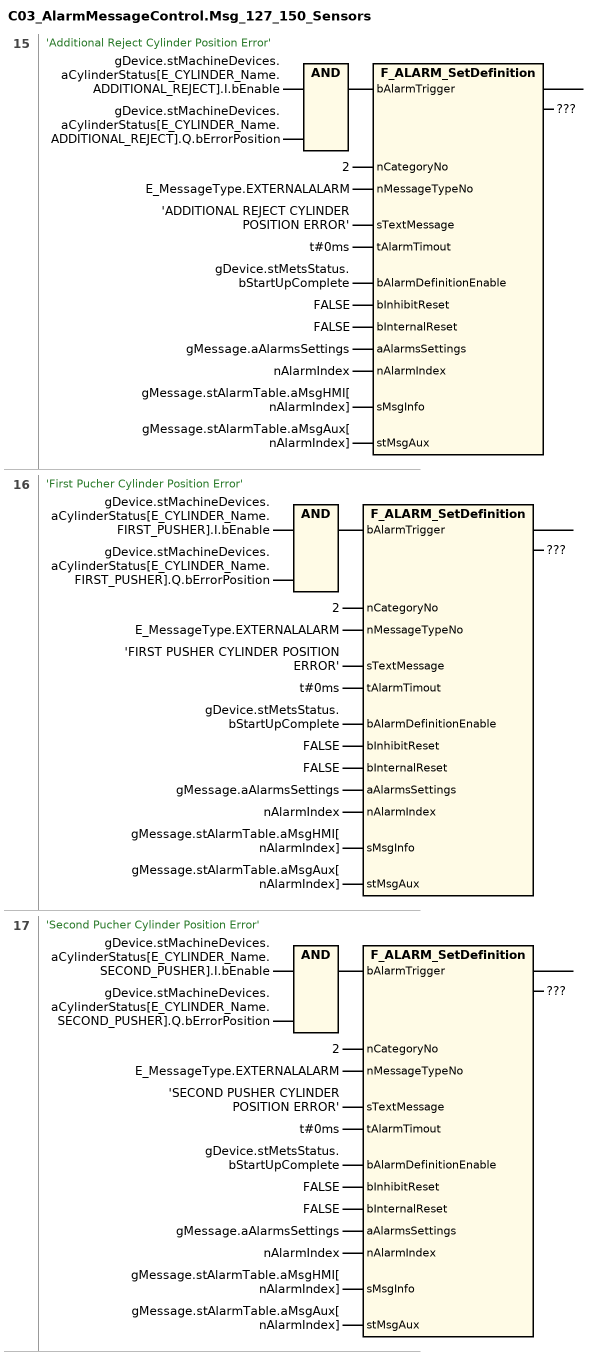
// NETWORK 15
// 'Additional Reject Cylinder Position Error'
F_ALARM_SetDefinition(bAlarmTrigger := gDevice.stMachineDevices.aCylinderStatus[E_CYLINDER_Name.ADDITIONAL_REJECT].I.bEnable AND gDevice.stMachineDevices.aCylinderStatus[E_CYLINDER_Name.ADDITIONAL_REJECT].Q.bErrorPosition, nCategoryNo := 2, nMessageTypeNo := E_MessageType.EXTERNALALARM, sTextMessage := 'ADDITIONAL REJECT CYLINDER POSITION ERROR', tAlarmTimout := t#0ms, bAlarmDefinitionEnable := gDevice.stMetsStatus.bStartUpComplete, bInhibitReset := FALSE, bInternalReset := FALSE, aAlarmsSettings := gMessage.aAlarmsSettings, nAlarmIndex := nAlarmIndex, sMsgInfo := gMessage.stAlarmTable.aMsgHMI[nAlarmIndex], stMsgAux := gMessage.stAlarmTable.aMsgAux[nAlarmIndex]);

// NETWORK 16
// 'First Pucher Cylinder Position Error'
F_ALARM_SetDefinition(bAlarmTrigger := gDevice.stMachineDevices.aCylinderStatus[E_CYLINDER_Name.FIRST_PUSHER].I.bEnable AND gDevice.stMachineDevices.aCylinderStatus[E_CYLINDER_Name.FIRST_PUSHER].Q.bErrorPosition, nCategoryNo := 2, nMessageTypeNo := E_MessageType.EXTERNALALARM, sTextMessage := 'FIRST PUSHER CYLINDER POSITION ERROR', tAlarmTimout := t#0ms, bAlarmDefinitionEnable := gDevice.stMetsStatus.bStartUpComplete, bInhibitReset := FALSE, bInternalReset := FALSE, aAlarmsSettings := gMessage.aAlarmsSettings, nAlarmIndex := nAlarmIndex, sMsgInfo := gMessage.stAlarmTable.aMsgHMI[nAlarmIndex], stMsgAux := gMessage.stAlarmTable.aMsgAux[nAlarmIndex]);

// NETWORK 17
// 'Second Pucher Cylinder Position Error'
F_ALARM_SetDefinition(bAlarmTrigger := gDevice.stMachineDevices.aCylinderStatus[E_CYLINDER_Name.SECOND_PUSHER].I.bEnable AND gDevice.stMachineDevices.aCylinderStatus[E_CYLINDER_Name.SECOND_PUSHER].Q.bErrorPosition, nCategoryNo := 2, nMessageTypeNo := E_MessageType.EXTERNALALARM, sTextMessage := 'SECOND PUSHER CYLINDER POSITION ERROR', tAlarmTimout := t#0ms, bAlarmDefinitionEnable := gDevice.stMetsStatus.bStartUpComplete, bInhibitReset := FALSE, bInternalReset := FALSE, aAlarmsSettings := gMessage.aAlarmsSettings, nAlarmIndex := nAlarmIndex, sMsgInfo := gMessage.stAlarmTable.aMsgHMI[nAlarmIndex], stMsgAux := gMessage.stAlarmTable.aMsgAux[nAlarmIndex]);

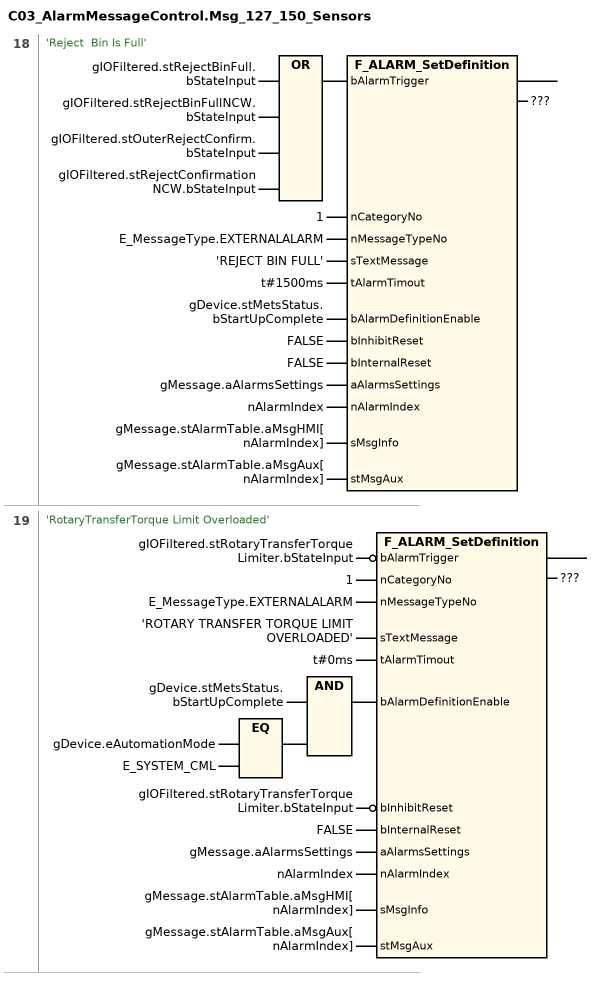
// NETWORK 18
// 'Reject  Bin Is Full'
F_ALARM_SetDefinition(bAlarmTrigger := gIOFiltered.stRejectBinFull.bStateInput OR gIOFiltered.stRejectBinFullNCW.bStateInput OR gIOFiltered.stOuterRejectConfirm.bStateInput OR gIOFiltered.stRejectConfirmationNCW.bStateInput, nCategoryNo := 1, nMessageTypeNo := E_MessageType.EXTERNALALARM, sTextMessage := 'REJECT BIN FULL', tAlarmTimout := t#1500ms, bAlarmDefinitionEnable := gDevice.stMetsStatus.bStartUpComplete, bInhibitReset := FALSE, bInternalReset := FALSE, aAlarmsSettings := gMessage.aAlarmsSettings, nAlarmIndex := nAlarmIndex, sMsgInfo := gMessage.stAlarmTable.aMsgHMI[nAlarmIndex], stMsgAux := gMessage.stAlarmTable.aMsgAux[nAlarmIndex]);

// NETWORK 19
// 'RotaryTransferTorque Limit Overloaded'
F_ALARM_SetDefinition(bAlarmTrigger := NOT gIOFiltered.stRotaryTransferTorqueLimiter.bStateInput, nCategoryNo := 1, nMessageTypeNo := E_MessageType.EXTERNALALARM, sTextMessage := 'ROTARY TRANSFER TORQUE LIMIT OVERLOADED', tAlarmTimout := t#0ms, bAlarmDefinitionEnable := gDevice.stMetsStatus.bStartUpComplete AND gDevice.eAutomationMode = E_SYSTEM_CML, bInhibitReset := NOT gIOFiltered.stRotaryTransferTorqueLimiter.bStateInput, bInternalReset := FALSE, aAlarmsSettings := gMessage.aAlarmsSettings, nAlarmIndex := nAlarmIndex, sMsgInfo := gMessage.stAlarmTable.aMsgHMI[nAlarmIndex], stMsgAux := gMessage.stAlarmTable.aMsgAux[nAlarmIndex]);

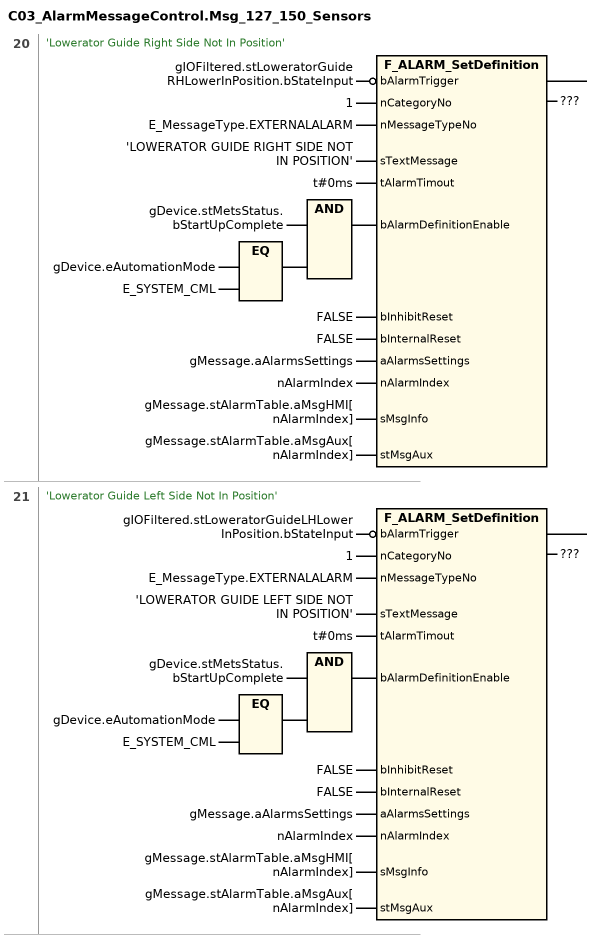
// NETWORK 20
// 'Lowerator Guide Right Side Not In Position'
F_ALARM_SetDefinition(bAlarmTrigger := NOT gIOFiltered.stLoweratorGuideRHLowerInPosition.bStateInput, nCategoryNo := 1, nMessageTypeNo := E_MessageType.EXTERNALALARM, sTextMessage := 'LOWERATOR GUIDE RIGHT SIDE NOT IN POSITION', tAlarmTimout := t#0ms, bAlarmDefinitionEnable := gDevice.stMetsStatus.bStartUpComplete AND gDevice.eAutomationMode = E_SYSTEM_CML, bInhibitReset := FALSE, bInternalReset := FALSE, aAlarmsSettings := gMessage.aAlarmsSettings, nAlarmIndex := nAlarmIndex, sMsgInfo := gMessage.stAlarmTable.aMsgHMI[nAlarmIndex], stMsgAux := gMessage.stAlarmTable.aMsgAux[nAlarmIndex]);

// NETWORK 21
// 'Lowerator Guide Left Side Not In Position'
F_ALARM_SetDefinition(bAlarmTrigger := NOT gIOFiltered.stLoweratorGuideLHLowerInPosition.bStateInput, nCategoryNo := 1, nMessageTypeNo := E_MessageType.EXTERNALALARM, sTextMessage := 'LOWERATOR GUIDE LEFT SIDE NOT IN POSITION', tAlarmTimout := t#0ms, bAlarmDefinitionEnable := gDevice.stMetsStatus.bStartUpComplete AND gDevice.eAutomationMode = E_SYSTEM_CML, bInhibitReset := FALSE, bInternalReset := FALSE, aAlarmsSettings := gMessage.aAlarmsSettings, nAlarmIndex := nAlarmIndex, sMsgInfo := gMessage.stAlarmTable.aMsgHMI[nAlarmIndex], stMsgAux := gMessage.stAlarmTable.aMsgAux[nAlarmIndex]);

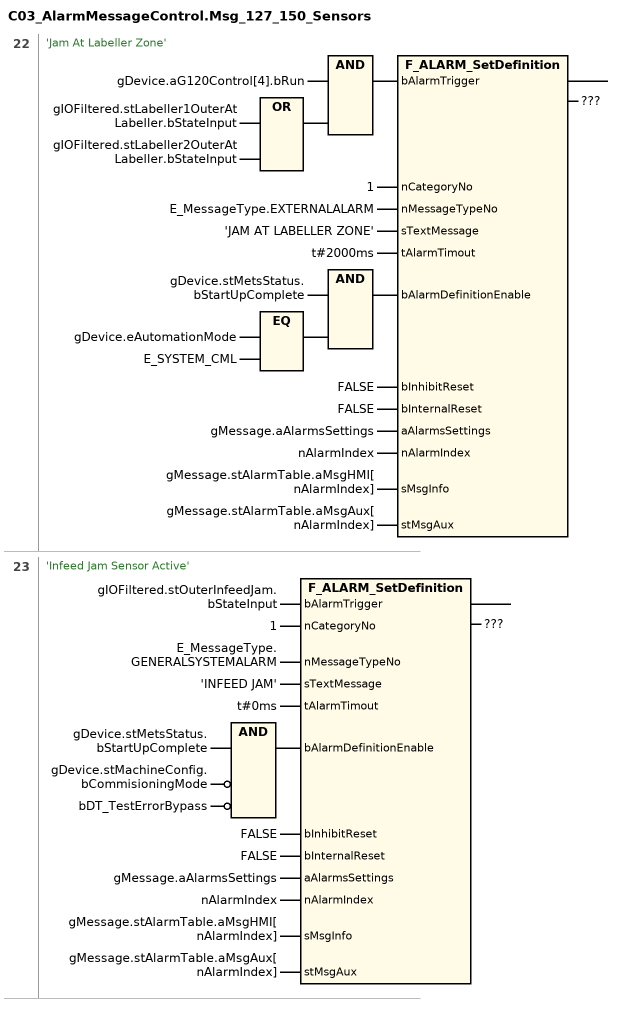
// NETWORK 22
// 'Jam At Labeller Zone'
F_ALARM_SetDefinition(bAlarmTrigger := gDevice.aG120Control[4].bRun AND (gIOFiltered.stLabeller1OuterAtLabeller.bStateInput OR gIOFiltered.stLabeller2OuterAtLabeller.bStateInput), nCategoryNo := 1, nMessageTypeNo := E_MessageType.EXTERNALALARM, sTextMessage := 'JAM AT LABELLER ZONE', tAlarmTimout := t#2000ms, bAlarmDefinitionEnable := gDevice.stMetsStatus.bStartUpComplete AND gDevice.eAutomationMode = E_SYSTEM_CML, bInhibitReset := FALSE, bInternalReset := FALSE, aAlarmsSettings := gMessage.aAlarmsSettings, nAlarmIndex := nAlarmIndex, sMsgInfo := gMessage.stAlarmTable.aMsgHMI[nAlarmIndex], stMsgAux := gMessage.stAlarmTable.aMsgAux[nAlarmIndex]);

// NETWORK 23
// 'Infeed Jam Sensor Active'
F_ALARM_SetDefinition(bAlarmTrigger := gIOFiltered.stOuterInfeedJam.bStateInput, nCategoryNo := 1, nMessageTypeNo := E_MessageType.GENERALSYSTEMALARM, sTextMessage := 'INFEED JAM', tAlarmTimout := t#0ms, bAlarmDefinitionEnable := gDevice.stMetsStatus.bStartUpComplete AND NOT gDevice.stMachineConfig.bCommisioningMode AND NOT bDT_TestErrorBypass, bInhibitReset := FALSE, bInternalReset := FALSE, aAlarmsSettings := gMessage.aAlarmsSettings, nAlarmIndex := nAlarmIndex, sMsgInfo := gMessage.stAlarmTable.aMsgHMI[nAlarmIndex], stMsgAux := gMessage.stAlarmTable.aMsgAux[nAlarmIndex]);

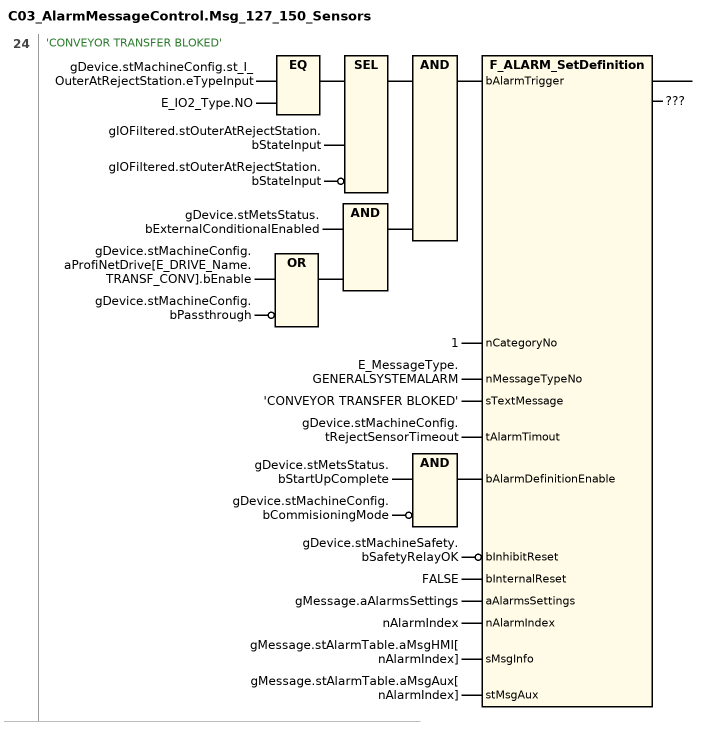
// NETWORK 24
// 'CONVEYOR TRANSFER BLOKED'
F_ALARM_SetDefinition(bAlarmTrigger := SEL(gDevice.stMachineConfig.st_I_OuterAtRejectStation.eTypeInput = E_IO2_Type.NO, gIOFiltered.stOuterAtRejectStation.bStateInput, NOT gIOFiltered.stOuterAtRejectStation.bStateInput) AND (gDevice.stMetsStatus.bExternalConditionalEnabled AND (gDevice.stMachineConfig.aProfiNetDrive[E_DRIVE_Name.TRANSF_CONV].bEnable OR NOT gDevice.stMachineConfig.bPassthrough)), nCategoryNo := 1, nMessageTypeNo := E_MessageType.GENERALSYSTEMALARM, sTextMessage := 'CONVEYOR TRANSFER BLOKED', tAlarmTimout := gDevice.stMachineConfig.tRejectSensorTimeout, bAlarmDefinitionEnable := gDevice.stMetsStatus.bStartUpComplete AND NOT gDevice.stMachineConfig.bCommisioningMode, bInhibitReset := NOT gDevice.stMachineSafety.bSafetyRelayOK, bInternalReset := FALSE, aAlarmsSettings := gMessage.aAlarmsSettings, nAlarmIndex := nAlarmIndex, sMsgInfo := gMessage.stAlarmTable.aMsgHMI[nAlarmIndex], stMsgAux := gMessage.stAlarmTable.aMsgAux[nAlarmIndex]);
END_ACTION

ACTION Msg_151_179_Doors:
// note: this text did not pass the execution check against the stored diagram
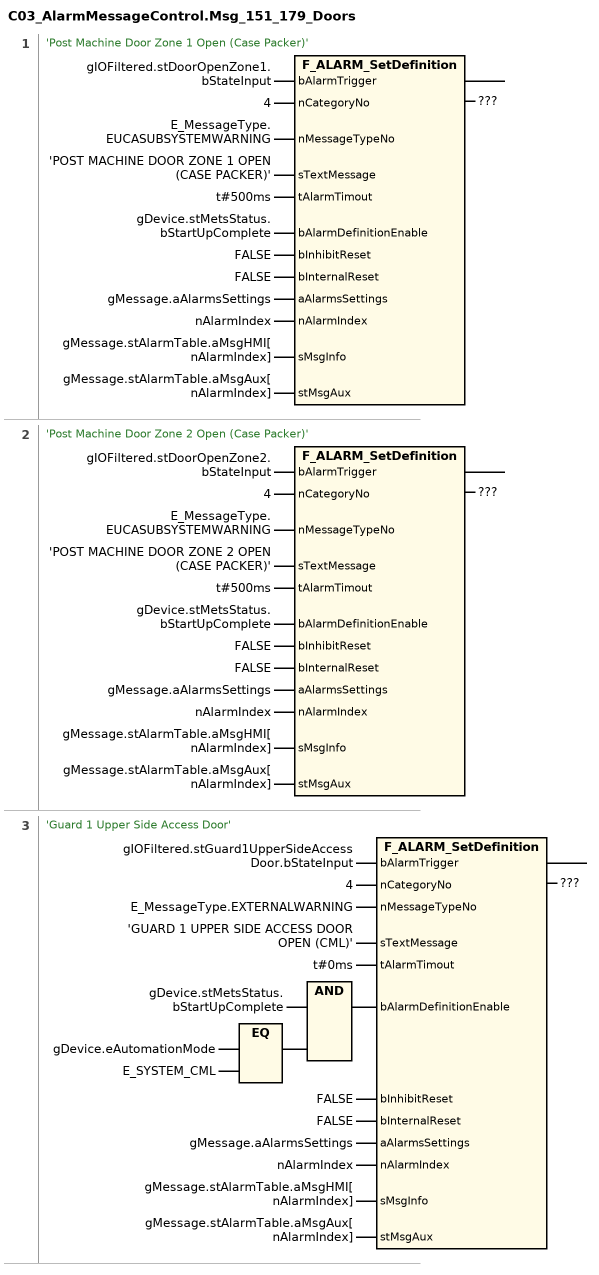
// NETWORK 1
// 'Post Machine Door Zone 1 Open (Case Packer)'
F_ALARM_SetDefinition(bAlarmTrigger := gIOFiltered.stDoorOpenZone1.bStateInput, nCategoryNo := 4, nMessageTypeNo := E_MessageType.EUCASUBSYSTEMWARNING, sTextMessage := 'POST MACHINE DOOR ZONE 1 OPEN (CASE PACKER)', tAlarmTimout := t#500ms, bAlarmDefinitionEnable := gDevice.stMetsStatus.bStartUpComplete, bInhibitReset := FALSE, bInternalReset := FALSE, aAlarmsSettings := gMessage.aAlarmsSettings, nAlarmIndex := nAlarmIndex, sMsgInfo := gMessage.stAlarmTable.aMsgHMI[nAlarmIndex], stMsgAux := gMessage.stAlarmTable.aMsgAux[nAlarmIndex]);

// NETWORK 2
// 'Post Machine Door Zone 2 Open (Case Packer)'
F_ALARM_SetDefinition(bAlarmTrigger := gIOFiltered.stDoorOpenZone2.bStateInput, nCategoryNo := 4, nMessageTypeNo := E_MessageType.EUCASUBSYSTEMWARNING, sTextMessage := 'POST MACHINE DOOR ZONE 2 OPEN (CASE PACKER)', tAlarmTimout := t#500ms, bAlarmDefinitionEnable := gDevice.stMetsStatus.bStartUpComplete, bInhibitReset := FALSE, bInternalReset := FALSE, aAlarmsSettings := gMessage.aAlarmsSettings, nAlarmIndex := nAlarmIndex, sMsgInfo := gMessage.stAlarmTable.aMsgHMI[nAlarmIndex], stMsgAux := gMessage.stAlarmTable.aMsgAux[nAlarmIndex]);

// NETWORK 3
// 'Guard 1 Upper Side Access Door'
F_ALARM_SetDefinition(bAlarmTrigger := gIOFiltered.stGuard1UpperSideAccessDoor.bStateInput, nCategoryNo := 4, nMessageTypeNo := E_MessageType.EXTERNALWARNING, sTextMessage := 'GUARD 1 UPPER SIDE ACCESS DOOR OPEN (CML)', tAlarmTimout := t#0ms, bAlarmDefinitionEnable := gDevice.stMetsStatus.bStartUpComplete AND gDevice.eAutomationMode = E_SYSTEM_CML, bInhibitReset := FALSE, bInternalReset := FALSE, aAlarmsSettings := gMessage.aAlarmsSettings, nAlarmIndex := nAlarmIndex, sMsgInfo := gMessage.stAlarmTable.aMsgHMI[nAlarmIndex], stMsgAux := gMessage.stAlarmTable.aMsgAux[nAlarmIndex]);

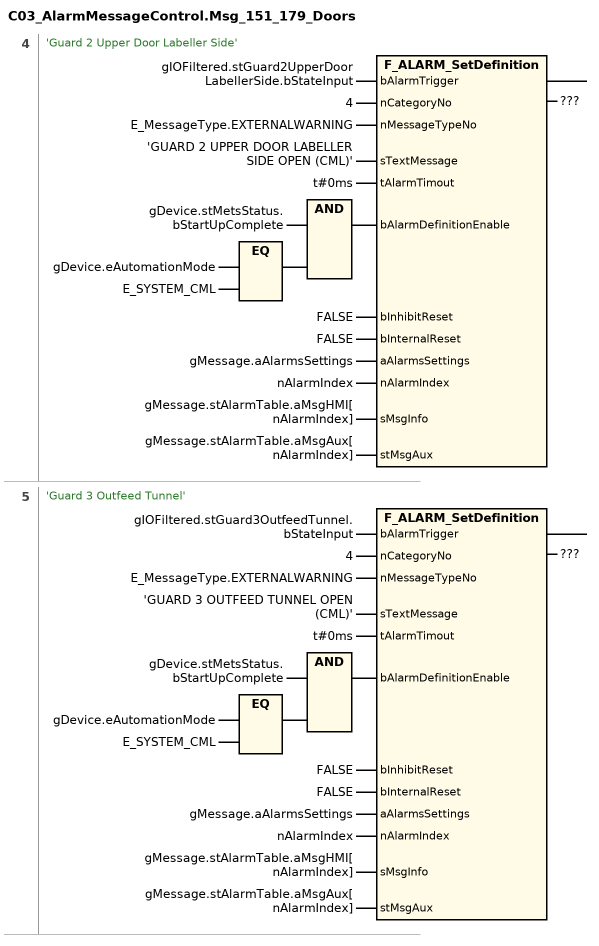
// NETWORK 4
// 'Guard 2 Upper Door Labeller Side'
F_ALARM_SetDefinition(bAlarmTrigger := gIOFiltered.stGuard2UpperDoorLabellerSide.bStateInput, nCategoryNo := 4, nMessageTypeNo := E_MessageType.EXTERNALWARNING, sTextMessage := 'GUARD 2 UPPER DOOR LABELLER SIDE OPEN (CML)', tAlarmTimout := t#0ms, bAlarmDefinitionEnable := gDevice.stMetsStatus.bStartUpComplete AND gDevice.eAutomationMode = E_SYSTEM_CML, bInhibitReset := FALSE, bInternalReset := FALSE, aAlarmsSettings := gMessage.aAlarmsSettings, nAlarmIndex := nAlarmIndex, sMsgInfo := gMessage.stAlarmTable.aMsgHMI[nAlarmIndex], stMsgAux := gMessage.stAlarmTable.aMsgAux[nAlarmIndex]);

// NETWORK 5
// 'Guard 3 Outfeed Tunnel'
F_ALARM_SetDefinition(bAlarmTrigger := gIOFiltered.stGuard3OutfeedTunnel.bStateInput, nCategoryNo := 4, nMessageTypeNo := E_MessageType.EXTERNALWARNING, sTextMessage := 'GUARD 3 OUTFEED TUNNEL OPEN (CML)', tAlarmTimout := t#0ms, bAlarmDefinitionEnable := gDevice.stMetsStatus.bStartUpComplete AND gDevice.eAutomationMode = E_SYSTEM_CML, bInhibitReset := FALSE, bInternalReset := FALSE, aAlarmsSettings := gMessage.aAlarmsSettings, nAlarmIndex := nAlarmIndex, sMsgInfo := gMessage.stAlarmTable.aMsgHMI[nAlarmIndex], stMsgAux := gMessage.stAlarmTable.aMsgAux[nAlarmIndex]);

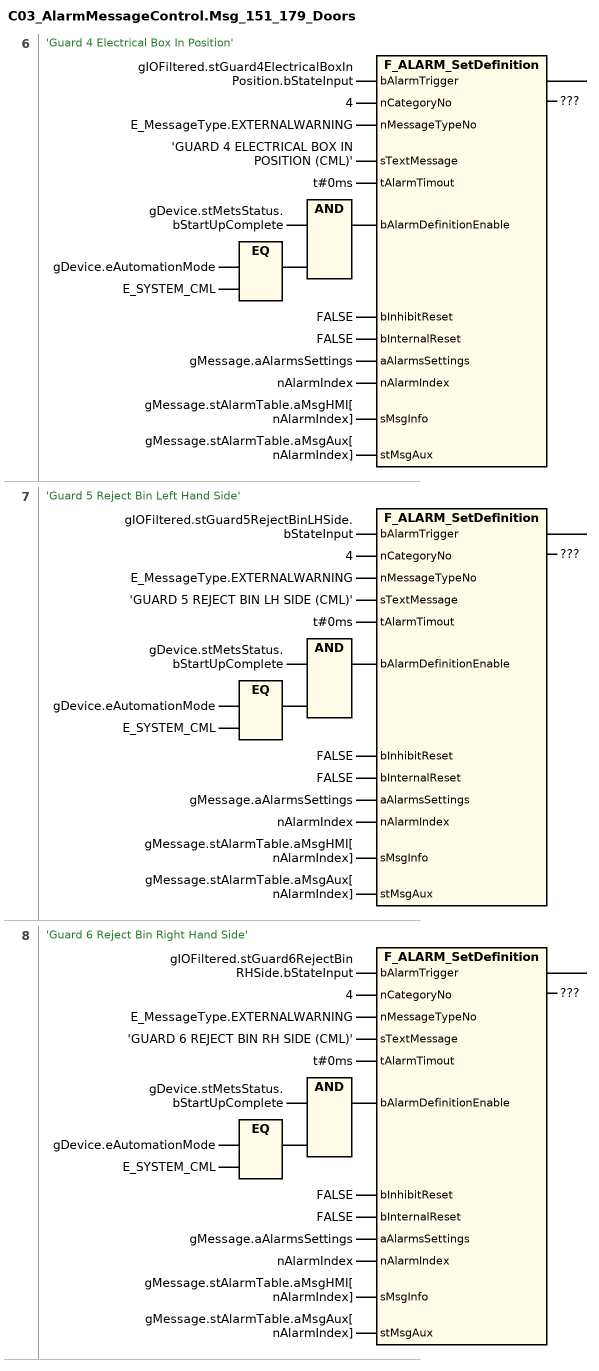
// NETWORK 6
// 'Guard 4 Electrical Box In Position'
F_ALARM_SetDefinition(bAlarmTrigger := gIOFiltered.stGuard4ElectricalBoxInPosition.bStateInput, nCategoryNo := 4, nMessageTypeNo := E_MessageType.EXTERNALWARNING, sTextMessage := 'GUARD 4 ELECTRICAL BOX IN POSITION (CML)', tAlarmTimout := t#0ms, bAlarmDefinitionEnable := gDevice.stMetsStatus.bStartUpComplete AND gDevice.eAutomationMode = E_SYSTEM_CML, bInhibitReset := FALSE, bInternalReset := FALSE, aAlarmsSettings := gMessage.aAlarmsSettings, nAlarmIndex := nAlarmIndex, sMsgInfo := gMessage.stAlarmTable.aMsgHMI[nAlarmIndex], stMsgAux := gMessage.stAlarmTable.aMsgAux[nAlarmIndex]);

// NETWORK 7
// 'Guard 5 Reject Bin Left Hand Side'
F_ALARM_SetDefinition(bAlarmTrigger := gIOFiltered.stGuard5RejectBinLHSide.bStateInput, nCategoryNo := 4, nMessageTypeNo := E_MessageType.EXTERNALWARNING, sTextMessage := 'GUARD 5 REJECT BIN LH SIDE (CML)', tAlarmTimout := t#0ms, bAlarmDefinitionEnable := gDevice.stMetsStatus.bStartUpComplete AND gDevice.eAutomationMode = E_SYSTEM_CML, bInhibitReset := FALSE, bInternalReset := FALSE, aAlarmsSettings := gMessage.aAlarmsSettings, nAlarmIndex := nAlarmIndex, sMsgInfo := gMessage.stAlarmTable.aMsgHMI[nAlarmIndex], stMsgAux := gMessage.stAlarmTable.aMsgAux[nAlarmIndex]);

// NETWORK 8
// 'Guard 6 Reject Bin Right Hand Side'
F_ALARM_SetDefinition(bAlarmTrigger := gIOFiltered.stGuard6RejectBinRHSide.bStateInput, nCategoryNo := 4, nMessageTypeNo := E_MessageType.EXTERNALWARNING, sTextMessage := 'GUARD 6 REJECT BIN RH SIDE (CML)', tAlarmTimout := t#0ms, bAlarmDefinitionEnable := gDevice.stMetsStatus.bStartUpComplete AND gDevice.eAutomationMode = E_SYSTEM_CML, bInhibitReset := FALSE, bInternalReset := FALSE, aAlarmsSettings := gMessage.aAlarmsSettings, nAlarmIndex := nAlarmIndex, sMsgInfo := gMessage.stAlarmTable.aMsgHMI[nAlarmIndex], stMsgAux := gMessage.stAlarmTable.aMsgAux[nAlarmIndex]);

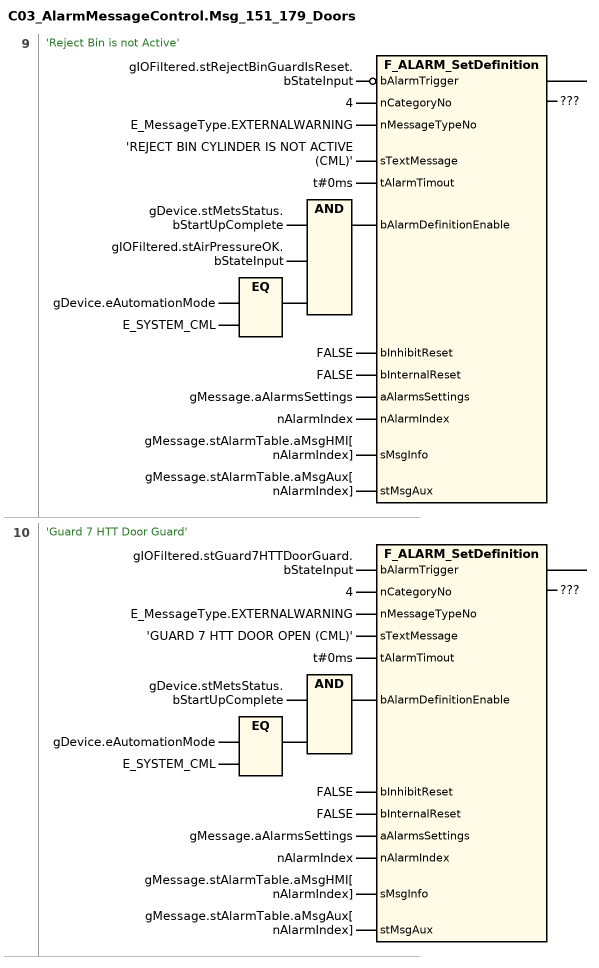
// NETWORK 9
// 'Reject Bin is not Active'
F_ALARM_SetDefinition(bAlarmTrigger := NOT gIOFiltered.stRejectBinGuardIsReset.bStateInput, nCategoryNo := 4, nMessageTypeNo := E_MessageType.EXTERNALWARNING, sTextMessage := 'REJECT BIN CYLINDER IS NOT ACTIVE (CML)', tAlarmTimout := t#0ms, bAlarmDefinitionEnable := gDevice.stMetsStatus.bStartUpComplete AND gIOFiltered.stAirPressureOK.bStateInput AND gDevice.eAutomationMode = E_SYSTEM_CML, bInhibitReset := FALSE, bInternalReset := FALSE, aAlarmsSettings := gMessage.aAlarmsSettings, nAlarmIndex := nAlarmIndex, sMsgInfo := gMessage.stAlarmTable.aMsgHMI[nAlarmIndex], stMsgAux := gMessage.stAlarmTable.aMsgAux[nAlarmIndex]);

// NETWORK 10
// 'Guard 7 HTT Door Guard'
F_ALARM_SetDefinition(bAlarmTrigger := gIOFiltered.stGuard7HTTDoorGuard.bStateInput, nCategoryNo := 4, nMessageTypeNo := E_MessageType.EXTERNALWARNING, sTextMessage := 'GUARD 7 HTT DOOR OPEN (CML)', tAlarmTimout := t#0ms, bAlarmDefinitionEnable := gDevice.stMetsStatus.bStartUpComplete AND gDevice.eAutomationMode = E_SYSTEM_CML, bInhibitReset := FALSE, bInternalReset := FALSE, aAlarmsSettings := gMessage.aAlarmsSettings, nAlarmIndex := nAlarmIndex, sMsgInfo := gMessage.stAlarmTable.aMsgHMI[nAlarmIndex], stMsgAux := gMessage.stAlarmTable.aMsgAux[nAlarmIndex]);

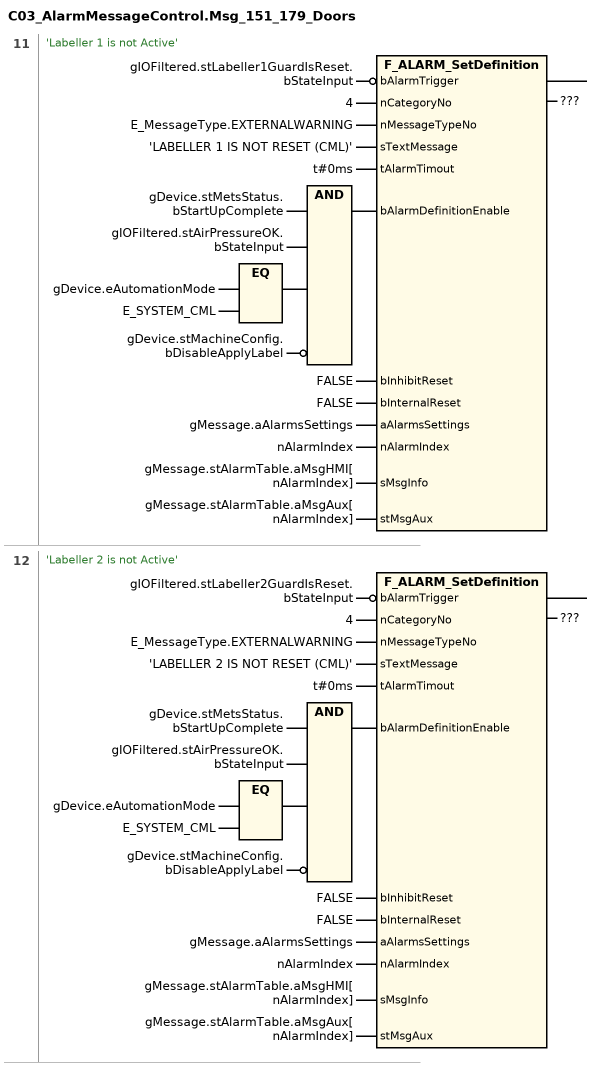
// NETWORK 11
// 'Labeller 1 is not Active'
F_ALARM_SetDefinition(bAlarmTrigger := NOT gIOFiltered.stLabeller1GuardIsReset.bStateInput, nCategoryNo := 4, nMessageTypeNo := E_MessageType.EXTERNALWARNING, sTextMessage := 'LABELLER 1 IS NOT RESET (CML)', tAlarmTimout := t#0ms, bAlarmDefinitionEnable := gDevice.stMetsStatus.bStartUpComplete AND gIOFiltered.stAirPressureOK.bStateInput AND gDevice.eAutomationMode = E_SYSTEM_CML AND NOT gDevice.stMachineConfig.bDisableApplyLabel, bInhibitReset := FALSE, bInternalReset := FALSE, aAlarmsSettings := gMessage.aAlarmsSettings, nAlarmIndex := nAlarmIndex, sMsgInfo := gMessage.stAlarmTable.aMsgHMI[nAlarmIndex], stMsgAux := gMessage.stAlarmTable.aMsgAux[nAlarmIndex]);

// NETWORK 12
// 'Labeller 2 is not Active'
F_ALARM_SetDefinition(bAlarmTrigger := NOT gIOFiltered.stLabeller2GuardIsReset.bStateInput, nCategoryNo := 4, nMessageTypeNo := E_MessageType.EXTERNALWARNING, sTextMessage := 'LABELLER 2 IS NOT RESET (CML)', tAlarmTimout := t#0ms, bAlarmDefinitionEnable := gDevice.stMetsStatus.bStartUpComplete AND gIOFiltered.stAirPressureOK.bStateInput AND gDevice.eAutomationMode = E_SYSTEM_CML AND NOT gDevice.stMachineConfig.bDisableApplyLabel, bInhibitReset := FALSE, bInternalReset := FALSE, aAlarmsSettings := gMessage.aAlarmsSettings, nAlarmIndex := nAlarmIndex, sMsgInfo := gMessage.stAlarmTable.aMsgHMI[nAlarmIndex], stMsgAux := gMessage.stAlarmTable.aMsgAux[nAlarmIndex]);

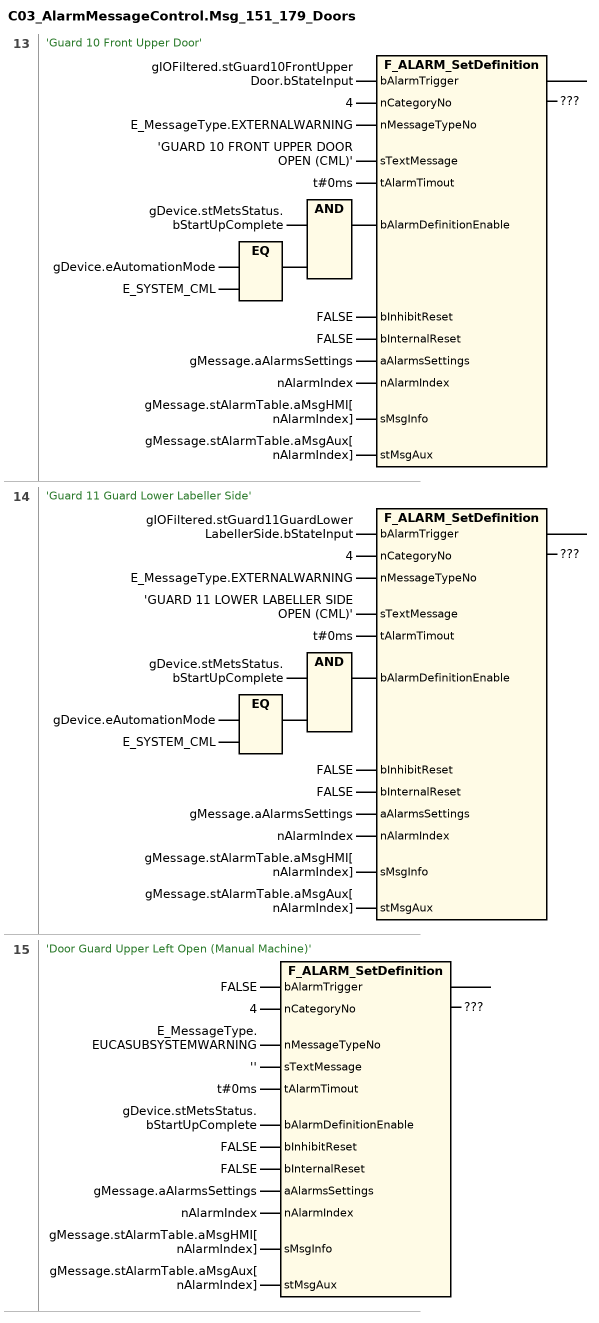
// NETWORK 13
// 'Guard 10 Front Upper Door'
F_ALARM_SetDefinition(bAlarmTrigger := gIOFiltered.stGuard10FrontUpperDoor.bStateInput, nCategoryNo := 4, nMessageTypeNo := E_MessageType.EXTERNALWARNING, sTextMessage := 'GUARD 10 FRONT UPPER DOOR OPEN (CML)', tAlarmTimout := t#0ms, bAlarmDefinitionEnable := gDevice.stMetsStatus.bStartUpComplete AND gDevice.eAutomationMode = E_SYSTEM_CML, bInhibitReset := FALSE, bInternalReset := FALSE, aAlarmsSettings := gMessage.aAlarmsSettings, nAlarmIndex := nAlarmIndex, sMsgInfo := gMessage.stAlarmTable.aMsgHMI[nAlarmIndex], stMsgAux := gMessage.stAlarmTable.aMsgAux[nAlarmIndex]);

// NETWORK 14
// 'Guard 11 Guard Lower Labeller Side'
F_ALARM_SetDefinition(bAlarmTrigger := gIOFiltered.stGuard11GuardLowerLabellerSide.bStateInput, nCategoryNo := 4, nMessageTypeNo := E_MessageType.EXTERNALWARNING, sTextMessage := 'GUARD 11 LOWER LABELLER SIDE OPEN (CML)', tAlarmTimout := t#0ms, bAlarmDefinitionEnable := gDevice.stMetsStatus.bStartUpComplete AND gDevice.eAutomationMode = E_SYSTEM_CML, bInhibitReset := FALSE, bInternalReset := FALSE, aAlarmsSettings := gMessage.aAlarmsSettings, nAlarmIndex := nAlarmIndex, sMsgInfo := gMessage.stAlarmTable.aMsgHMI[nAlarmIndex], stMsgAux := gMessage.stAlarmTable.aMsgAux[nAlarmIndex]);

// NETWORK 15
// 'Door Guard Upper Left Open (Manual Machine)'
F_ALARM_SetDefinition(bAlarmTrigger := FALSE, nCategoryNo := 4, nMessageTypeNo := E_MessageType.EUCASUBSYSTEMWARNING, sTextMessage := '', tAlarmTimout := t#0ms, bAlarmDefinitionEnable := gDevice.stMetsStatus.bStartUpComplete, bInhibitReset := FALSE, bInternalReset := FALSE, aAlarmsSettings := gMessage.aAlarmsSettings, nAlarmIndex := nAlarmIndex, sMsgInfo := gMessage.stAlarmTable.aMsgHMI[nAlarmIndex], stMsgAux := gMessage.stAlarmTable.aMsgAux[nAlarmIndex]);

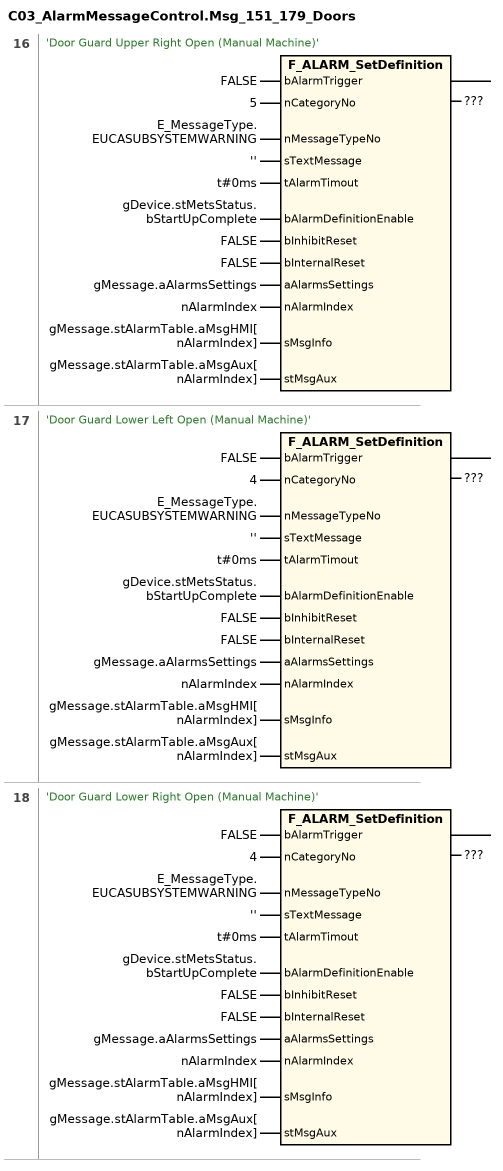
// NETWORK 16
// 'Door Guard Upper Right Open (Manual Machine)'
F_ALARM_SetDefinition(bAlarmTrigger := FALSE, nCategoryNo := 5, nMessageTypeNo := E_MessageType.EUCASUBSYSTEMWARNING, sTextMessage := '', tAlarmTimout := t#0ms, bAlarmDefinitionEnable := gDevice.stMetsStatus.bStartUpComplete, bInhibitReset := FALSE, bInternalReset := FALSE, aAlarmsSettings := gMessage.aAlarmsSettings, nAlarmIndex := nAlarmIndex, sMsgInfo := gMessage.stAlarmTable.aMsgHMI[nAlarmIndex], stMsgAux := gMessage.stAlarmTable.aMsgAux[nAlarmIndex]);

// NETWORK 17
// 'Door Guard Lower Left Open (Manual Machine)'
F_ALARM_SetDefinition(bAlarmTrigger := FALSE, nCategoryNo := 4, nMessageTypeNo := E_MessageType.EUCASUBSYSTEMWARNING, sTextMessage := '', tAlarmTimout := t#0ms, bAlarmDefinitionEnable := gDevice.stMetsStatus.bStartUpComplete, bInhibitReset := FALSE, bInternalReset := FALSE, aAlarmsSettings := gMessage.aAlarmsSettings, nAlarmIndex := nAlarmIndex, sMsgInfo := gMessage.stAlarmTable.aMsgHMI[nAlarmIndex], stMsgAux := gMessage.stAlarmTable.aMsgAux[nAlarmIndex]);

// NETWORK 18
// 'Door Guard Lower Right Open (Manual Machine)'
F_ALARM_SetDefinition(bAlarmTrigger := FALSE, nCategoryNo := 4, nMessageTypeNo := E_MessageType.EUCASUBSYSTEMWARNING, sTextMessage := '', tAlarmTimout := t#0ms, bAlarmDefinitionEnable := gDevice.stMetsStatus.bStartUpComplete, bInhibitReset := FALSE, bInternalReset := FALSE, aAlarmsSettings := gMessage.aAlarmsSettings, nAlarmIndex := nAlarmIndex, sMsgInfo := gMessage.stAlarmTable.aMsgHMI[nAlarmIndex], stMsgAux := gMessage.stAlarmTable.aMsgAux[nAlarmIndex]);

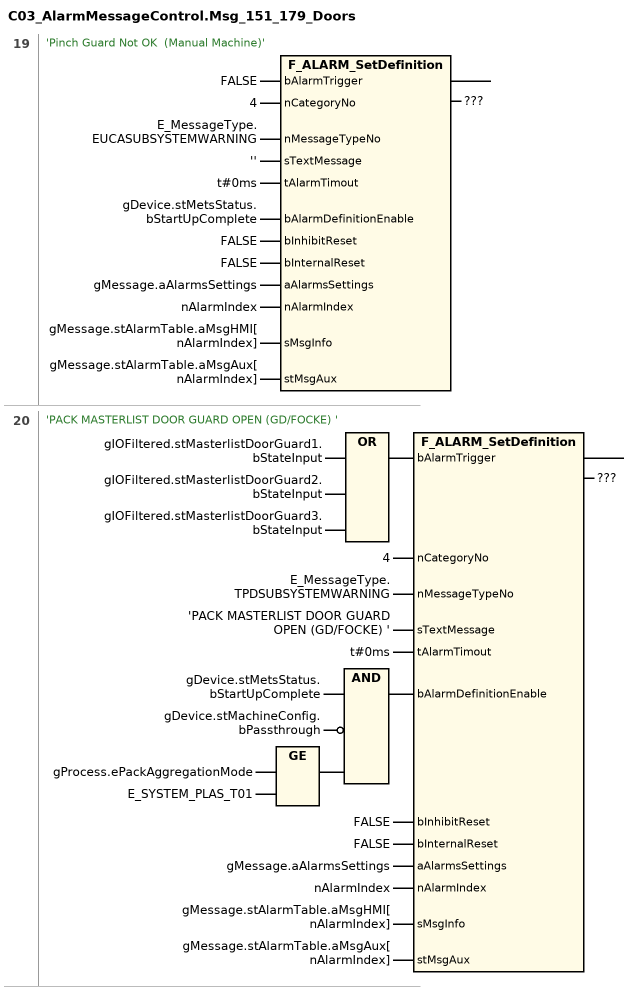
// NETWORK 19
// 'Pinch Guard Not OK  (Manual Machine)'
F_ALARM_SetDefinition(bAlarmTrigger := FALSE, nCategoryNo := 4, nMessageTypeNo := E_MessageType.EUCASUBSYSTEMWARNING, sTextMessage := '', tAlarmTimout := t#0ms, bAlarmDefinitionEnable := gDevice.stMetsStatus.bStartUpComplete, bInhibitReset := FALSE, bInternalReset := FALSE, aAlarmsSettings := gMessage.aAlarmsSettings, nAlarmIndex := nAlarmIndex, sMsgInfo := gMessage.stAlarmTable.aMsgHMI[nAlarmIndex], stMsgAux := gMessage.stAlarmTable.aMsgAux[nAlarmIndex]);

// NETWORK 20
// 'PACK MASTERLIST DOOR GUARD OPEN (GD/FOCKE) '
F_ALARM_SetDefinition(bAlarmTrigger := gIOFiltered.stMasterlistDoorGuard1.bStateInput OR gIOFiltered.stMasterlistDoorGuard2.bStateInput OR gIOFiltered.stMasterlistDoorGuard3.bStateInput, nCategoryNo := 4, nMessageTypeNo := E_MessageType.TPDSUBSYSTEMWARNING, sTextMessage := 'PACK MASTERLIST DOOR GUARD OPEN (GD/FOCKE) ', tAlarmTimout := t#0ms, bAlarmDefinitionEnable := gDevice.stMetsStatus.bStartUpComplete AND NOT gDevice.stMachineConfig.bPassthrough AND gProcess.ePackAggregationMode >= E_SYSTEM_PLAS_T01, bInhibitReset := FALSE, bInternalReset := FALSE, aAlarmsSettings := gMessage.aAlarmsSettings, nAlarmIndex := nAlarmIndex, sMsgInfo := gMessage.stAlarmTable.aMsgHMI[nAlarmIndex], stMsgAux := gMessage.stAlarmTable.aMsgAux[nAlarmIndex]);

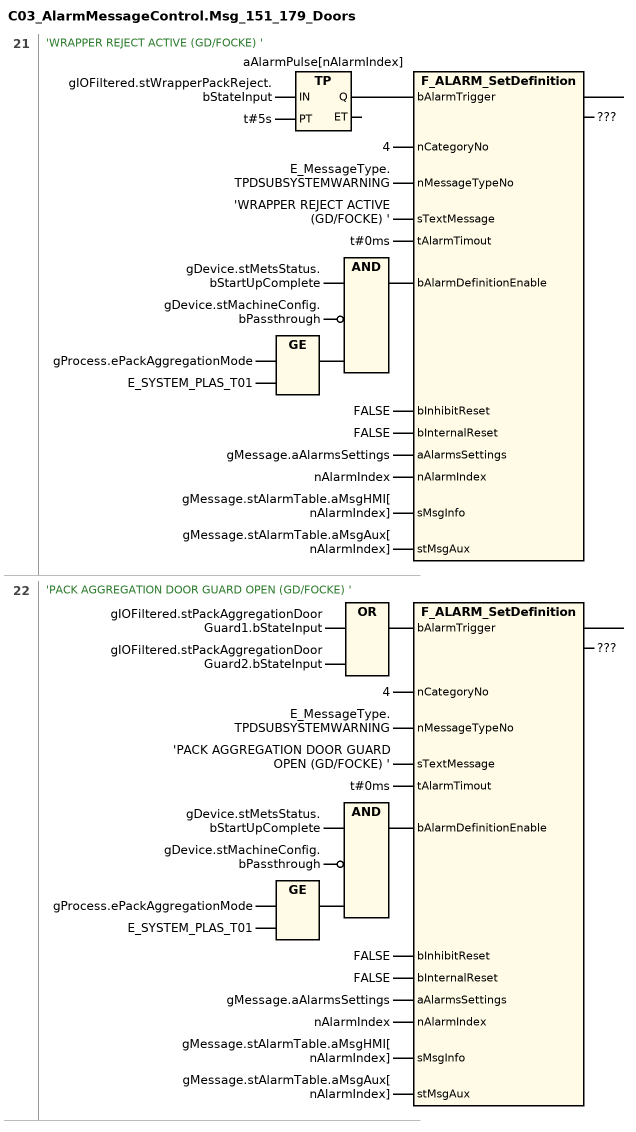
// NETWORK 21
// 'WRAPPER REJECT ACTIVE (GD/FOCKE) '
aAlarmPulse[nAlarmIndex](IN := gIOFiltered.stWrapperPackReject.bStateInput, PT := t#5s); // TP
F_ALARM_SetDefinition(bAlarmTrigger := aAlarmPulse[nAlarmIndex].Q, nCategoryNo := 4, nMessageTypeNo := E_MessageType.TPDSUBSYSTEMWARNING, sTextMessage := 'WRAPPER REJECT ACTIVE (GD/FOCKE) ', tAlarmTimout := t#0ms, bAlarmDefinitionEnable := gDevice.stMetsStatus.bStartUpComplete AND NOT gDevice.stMachineConfig.bPassthrough AND gProcess.ePackAggregationMode >= E_SYSTEM_PLAS_T01, bInhibitReset := FALSE, bInternalReset := FALSE, aAlarmsSettings := gMessage.aAlarmsSettings, nAlarmIndex := nAlarmIndex, sMsgInfo := gMessage.stAlarmTable.aMsgHMI[nAlarmIndex], stMsgAux := gMessage.stAlarmTable.aMsgAux[nAlarmIndex]);

// NETWORK 22
// 'PACK AGGREGATION DOOR GUARD OPEN (GD/FOCKE) '
F_ALARM_SetDefinition(bAlarmTrigger := gIOFiltered.stPackAggregationDoorGuard1.bStateInput OR gIOFiltered.stPackAggregationDoorGuard2.bStateInput, nCategoryNo := 4, nMessageTypeNo := E_MessageType.TPDSUBSYSTEMWARNING, sTextMessage := 'PACK AGGREGATION DOOR GUARD OPEN (GD/FOCKE) ', tAlarmTimout := t#0ms, bAlarmDefinitionEnable := gDevice.stMetsStatus.bStartUpComplete AND NOT gDevice.stMachineConfig.bPassthrough AND gProcess.ePackAggregationMode >= E_SYSTEM_PLAS_T01, bInhibitReset := FALSE, bInternalReset := FALSE, aAlarmsSettings := gMessage.aAlarmsSettings, nAlarmIndex := nAlarmIndex, sMsgInfo := gMessage.stAlarmTable.aMsgHMI[nAlarmIndex], stMsgAux := gMessage.stAlarmTable.aMsgAux[nAlarmIndex]);

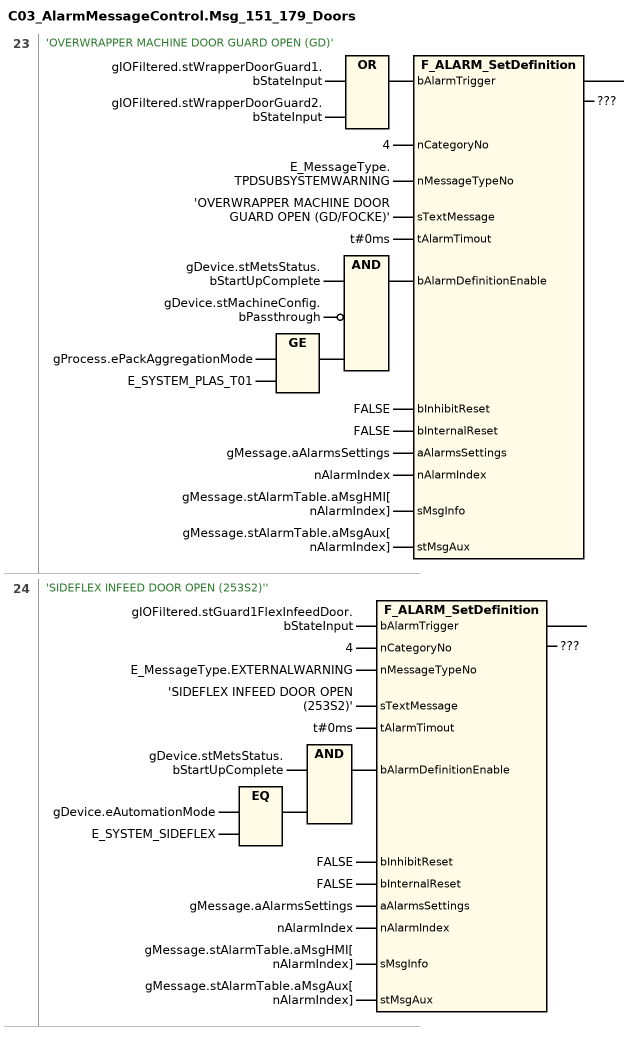
// NETWORK 23
// 'OVERWRAPPER MACHINE DOOR GUARD OPEN (GD)'
F_ALARM_SetDefinition(bAlarmTrigger := gIOFiltered.stWrapperDoorGuard1.bStateInput OR gIOFiltered.stWrapperDoorGuard2.bStateInput, nCategoryNo := 4, nMessageTypeNo := E_MessageType.TPDSUBSYSTEMWARNING, sTextMessage := 'OVERWRAPPER MACHINE DOOR GUARD OPEN (GD/FOCKE)', tAlarmTimout := t#0ms, bAlarmDefinitionEnable := gDevice.stMetsStatus.bStartUpComplete AND NOT gDevice.stMachineConfig.bPassthrough AND gProcess.ePackAggregationMode >= E_SYSTEM_PLAS_T01, bInhibitReset := FALSE, bInternalReset := FALSE, aAlarmsSettings := gMessage.aAlarmsSettings, nAlarmIndex := nAlarmIndex, sMsgInfo := gMessage.stAlarmTable.aMsgHMI[nAlarmIndex], stMsgAux := gMessage.stAlarmTable.aMsgAux[nAlarmIndex]);

// NETWORK 24
// 'SIDEFLEX INFEED DOOR OPEN (253S2)''
F_ALARM_SetDefinition(bAlarmTrigger := gIOFiltered.stGuard1FlexInfeedDoor.bStateInput, nCategoryNo := 4, nMessageTypeNo := E_MessageType.EXTERNALWARNING, sTextMessage := 'SIDEFLEX INFEED DOOR OPEN (253S2)', tAlarmTimout := t#0ms, bAlarmDefinitionEnable := gDevice.stMetsStatus.bStartUpComplete AND gDevice.eAutomationMode = E_SYSTEM_SIDEFLEX, bInhibitReset := FALSE, bInternalReset := FALSE, aAlarmsSettings := gMessage.aAlarmsSettings, nAlarmIndex := nAlarmIndex, sMsgInfo := gMessage.stAlarmTable.aMsgHMI[nAlarmIndex], stMsgAux := gMessage.stAlarmTable.aMsgAux[nAlarmIndex]);

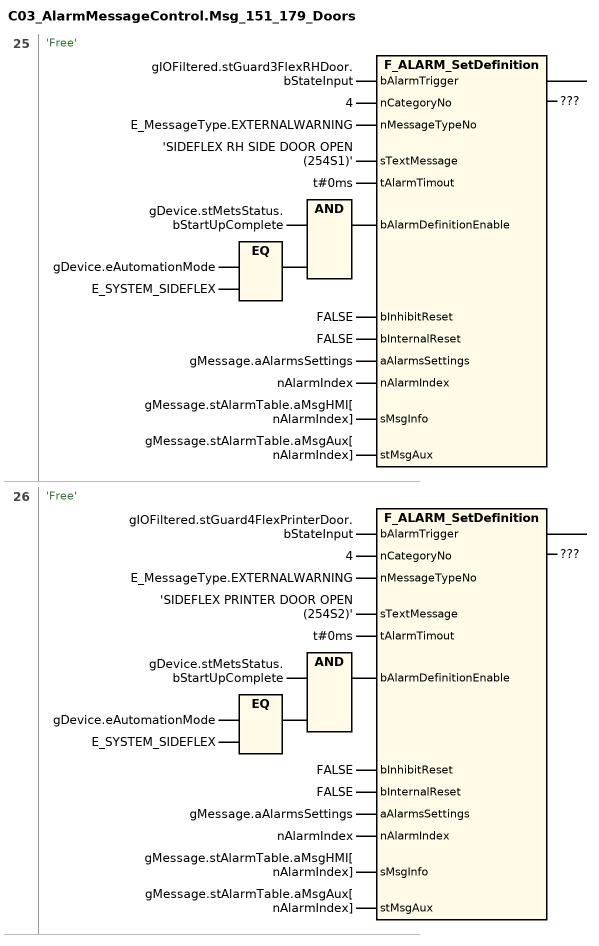
// NETWORK 25
// 'Free'
F_ALARM_SetDefinition(bAlarmTrigger := gIOFiltered.stGuard3FlexRHDoor.bStateInput, nCategoryNo := 4, nMessageTypeNo := E_MessageType.EXTERNALWARNING, sTextMessage := 'SIDEFLEX RH SIDE DOOR OPEN (254S1)', tAlarmTimout := t#0ms, bAlarmDefinitionEnable := gDevice.stMetsStatus.bStartUpComplete AND gDevice.eAutomationMode = E_SYSTEM_SIDEFLEX, bInhibitReset := FALSE, bInternalReset := FALSE, aAlarmsSettings := gMessage.aAlarmsSettings, nAlarmIndex := nAlarmIndex, sMsgInfo := gMessage.stAlarmTable.aMsgHMI[nAlarmIndex], stMsgAux := gMessage.stAlarmTable.aMsgAux[nAlarmIndex]);

// NETWORK 26
// 'Free'
F_ALARM_SetDefinition(bAlarmTrigger := gIOFiltered.stGuard4FlexPrinterDoor.bStateInput, nCategoryNo := 4, nMessageTypeNo := E_MessageType.EXTERNALWARNING, sTextMessage := 'SIDEFLEX PRINTER DOOR OPEN (254S2)', tAlarmTimout := t#0ms, bAlarmDefinitionEnable := gDevice.stMetsStatus.bStartUpComplete AND gDevice.eAutomationMode = E_SYSTEM_SIDEFLEX, bInhibitReset := FALSE, bInternalReset := FALSE, aAlarmsSettings := gMessage.aAlarmsSettings, nAlarmIndex := nAlarmIndex, sMsgInfo := gMessage.stAlarmTable.aMsgHMI[nAlarmIndex], stMsgAux := gMessage.stAlarmTable.aMsgAux[nAlarmIndex]);

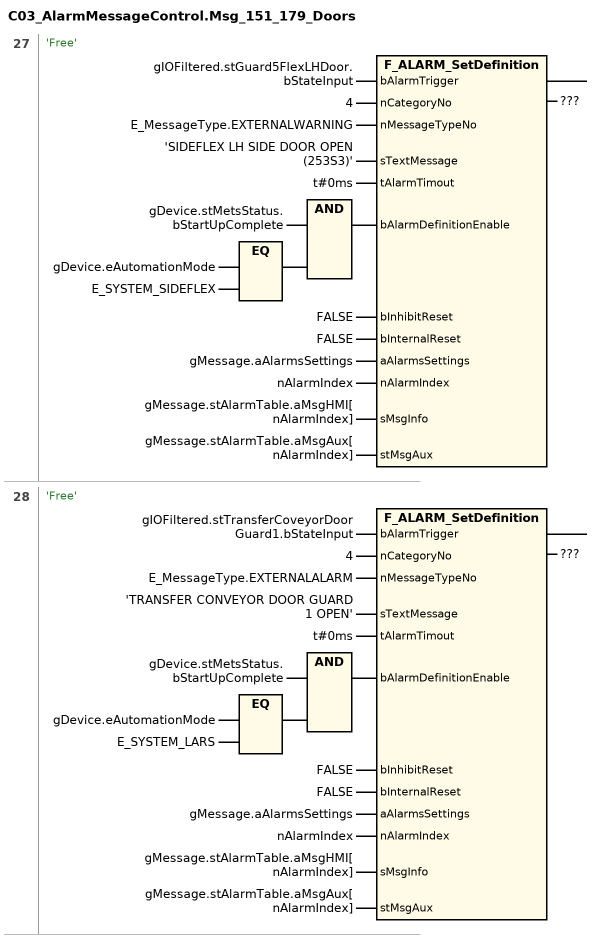
// NETWORK 27
// 'Free'
F_ALARM_SetDefinition(bAlarmTrigger := gIOFiltered.stGuard5FlexLHDoor.bStateInput, nCategoryNo := 4, nMessageTypeNo := E_MessageType.EXTERNALWARNING, sTextMessage := 'SIDEFLEX LH SIDE DOOR OPEN (253S3)', tAlarmTimout := t#0ms, bAlarmDefinitionEnable := gDevice.stMetsStatus.bStartUpComplete AND gDevice.eAutomationMode = E_SYSTEM_SIDEFLEX, bInhibitReset := FALSE, bInternalReset := FALSE, aAlarmsSettings := gMessage.aAlarmsSettings, nAlarmIndex := nAlarmIndex, sMsgInfo := gMessage.stAlarmTable.aMsgHMI[nAlarmIndex], stMsgAux := gMessage.stAlarmTable.aMsgAux[nAlarmIndex]);

// NETWORK 28
// 'Free'
F_ALARM_SetDefinition(bAlarmTrigger := gIOFiltered.stTransferCoveyorDoorGuard1.bStateInput, nCategoryNo := 4, nMessageTypeNo := E_MessageType.EXTERNALALARM, sTextMessage := 'TRANSFER CONVEYOR DOOR GUARD 1 OPEN', tAlarmTimout := t#0ms, bAlarmDefinitionEnable := gDevice.stMetsStatus.bStartUpComplete AND gDevice.eAutomationMode = E_SYSTEM_LARS, bInhibitReset := FALSE, bInternalReset := FALSE, aAlarmsSettings := gMessage.aAlarmsSettings, nAlarmIndex := nAlarmIndex, sMsgInfo := gMessage.stAlarmTable.aMsgHMI[nAlarmIndex], stMsgAux := gMessage.stAlarmTable.aMsgAux[nAlarmIndex]);

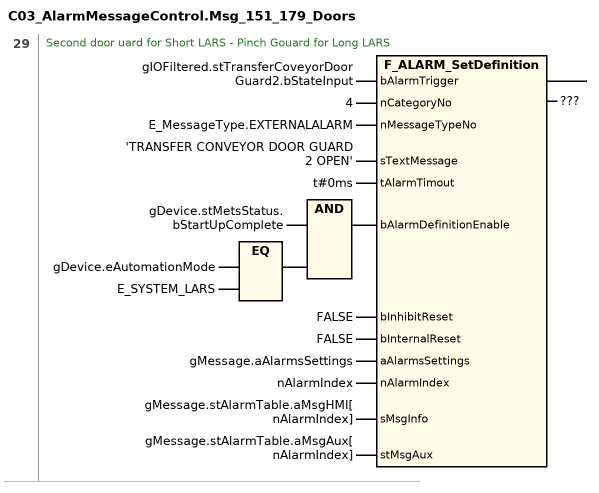
// NETWORK 29
// Second door uard for Short LARS - Pinch Gouard for Long LARS
F_ALARM_SetDefinition(bAlarmTrigger := gIOFiltered.stTransferCoveyorDoorGuard2.bStateInput, nCategoryNo := 4, nMessageTypeNo := E_MessageType.EXTERNALALARM, sTextMessage := 'TRANSFER CONVEYOR DOOR GUARD 2 OPEN', tAlarmTimout := t#0ms, bAlarmDefinitionEnable := gDevice.stMetsStatus.bStartUpComplete AND gDevice.eAutomationMode = E_SYSTEM_LARS, bInhibitReset := FALSE, bInternalReset := FALSE, aAlarmsSettings := gMessage.aAlarmsSettings, nAlarmIndex := nAlarmIndex, sMsgInfo := gMessage.stAlarmTable.aMsgHMI[nAlarmIndex], stMsgAux := gMessage.stAlarmTable.aMsgAux[nAlarmIndex]);
END_ACTION

ACTION Msg_180_200_Motors:
// note: this text did not pass the execution check against the stored diagram
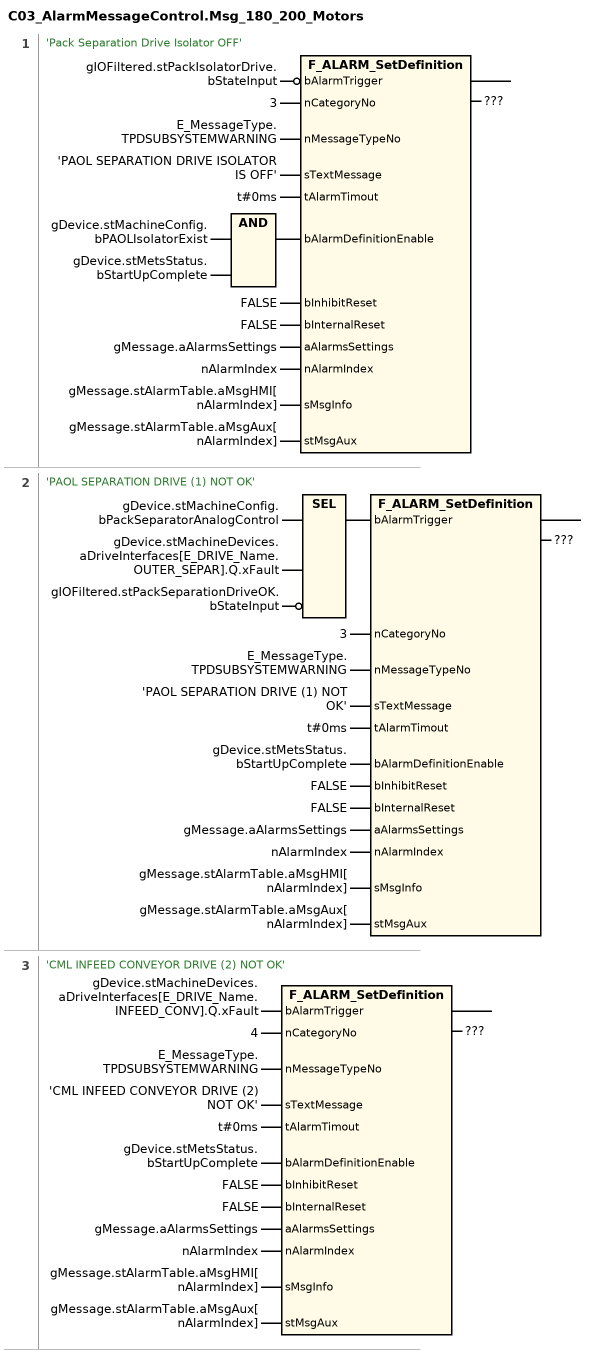
// NETWORK 1
// 'Pack Separation Drive Isolator OFF'
F_ALARM_SetDefinition(bAlarmTrigger := NOT gIOFiltered.stPackIsolatorDrive.bStateInput, nCategoryNo := 3, nMessageTypeNo := E_MessageType.TPDSUBSYSTEMWARNING, sTextMessage := 'PAOL SEPARATION DRIVE ISOLATOR IS OFF', tAlarmTimout := t#0ms, bAlarmDefinitionEnable := gDevice.stMachineConfig.bPAOLIsolatorExist AND gDevice.stMetsStatus.bStartUpComplete, bInhibitReset := FALSE, bInternalReset := FALSE, aAlarmsSettings := gMessage.aAlarmsSettings, nAlarmIndex := nAlarmIndex, sMsgInfo := gMessage.stAlarmTable.aMsgHMI[nAlarmIndex], stMsgAux := gMessage.stAlarmTable.aMsgAux[nAlarmIndex]);

// NETWORK 2
// 'PAOL SEPARATION DRIVE (1) NOT OK'
F_ALARM_SetDefinition(bAlarmTrigger := SEL(gDevice.stMachineConfig.bPackSeparatorAnalogControl, gDevice.stMachineDevices.aDriveInterfaces[E_DRIVE_Name.OUTER_SEPAR].Q.xFault, NOT gIOFiltered.stPackSeparationDriveOK.bStateInput), nCategoryNo := 3, nMessageTypeNo := E_MessageType.TPDSUBSYSTEMWARNING, sTextMessage := 'PAOL SEPARATION DRIVE (1) NOT OK', tAlarmTimout := t#0ms, bAlarmDefinitionEnable := gDevice.stMetsStatus.bStartUpComplete, bInhibitReset := FALSE, bInternalReset := FALSE, aAlarmsSettings := gMessage.aAlarmsSettings, nAlarmIndex := nAlarmIndex, sMsgInfo := gMessage.stAlarmTable.aMsgHMI[nAlarmIndex], stMsgAux := gMessage.stAlarmTable.aMsgAux[nAlarmIndex]);

// NETWORK 3
// 'CML INFEED CONVEYOR DRIVE (2) NOT OK'
F_ALARM_SetDefinition(bAlarmTrigger := gDevice.stMachineDevices.aDriveInterfaces[E_DRIVE_Name.INFEED_CONV].Q.xFault, nCategoryNo := 4, nMessageTypeNo := E_MessageType.TPDSUBSYSTEMWARNING, sTextMessage := 'CML INFEED CONVEYOR DRIVE (2) NOT OK', tAlarmTimout := t#0ms, bAlarmDefinitionEnable := gDevice.stMetsStatus.bStartUpComplete, bInhibitReset := FALSE, bInternalReset := FALSE, aAlarmsSettings := gMessage.aAlarmsSettings, nAlarmIndex := nAlarmIndex, sMsgInfo := gMessage.stAlarmTable.aMsgHMI[nAlarmIndex], stMsgAux := gMessage.stAlarmTable.aMsgAux[nAlarmIndex]);

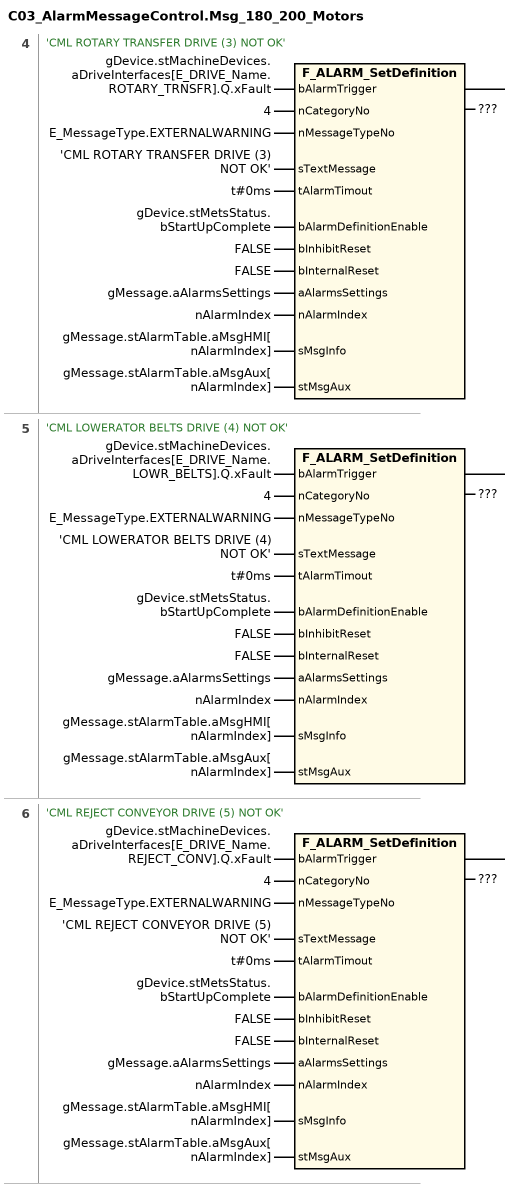
// NETWORK 4
// 'CML ROTARY TRANSFER DRIVE (3) NOT OK'
F_ALARM_SetDefinition(bAlarmTrigger := gDevice.stMachineDevices.aDriveInterfaces[E_DRIVE_Name.ROTARY_TRNSFR].Q.xFault, nCategoryNo := 4, nMessageTypeNo := E_MessageType.EXTERNALWARNING, sTextMessage := 'CML ROTARY TRANSFER DRIVE (3) NOT OK', tAlarmTimout := t#0ms, bAlarmDefinitionEnable := gDevice.stMetsStatus.bStartUpComplete, bInhibitReset := FALSE, bInternalReset := FALSE, aAlarmsSettings := gMessage.aAlarmsSettings, nAlarmIndex := nAlarmIndex, sMsgInfo := gMessage.stAlarmTable.aMsgHMI[nAlarmIndex], stMsgAux := gMessage.stAlarmTable.aMsgAux[nAlarmIndex]);

// NETWORK 5
// 'CML LOWERATOR BELTS DRIVE (4) NOT OK'
F_ALARM_SetDefinition(bAlarmTrigger := gDevice.stMachineDevices.aDriveInterfaces[E_DRIVE_Name.LOWR_BELTS].Q.xFault, nCategoryNo := 4, nMessageTypeNo := E_MessageType.EXTERNALWARNING, sTextMessage := 'CML LOWERATOR BELTS DRIVE (4) NOT OK', tAlarmTimout := t#0ms, bAlarmDefinitionEnable := gDevice.stMetsStatus.bStartUpComplete, bInhibitReset := FALSE, bInternalReset := FALSE, aAlarmsSettings := gMessage.aAlarmsSettings, nAlarmIndex := nAlarmIndex, sMsgInfo := gMessage.stAlarmTable.aMsgHMI[nAlarmIndex], stMsgAux := gMessage.stAlarmTable.aMsgAux[nAlarmIndex]);

// NETWORK 6
// 'CML REJECT CONVEYOR DRIVE (5) NOT OK'
F_ALARM_SetDefinition(bAlarmTrigger := gDevice.stMachineDevices.aDriveInterfaces[E_DRIVE_Name.REJECT_CONV].Q.xFault, nCategoryNo := 4, nMessageTypeNo := E_MessageType.EXTERNALWARNING, sTextMessage := 'CML REJECT CONVEYOR DRIVE (5) NOT OK', tAlarmTimout := t#0ms, bAlarmDefinitionEnable := gDevice.stMetsStatus.bStartUpComplete, bInhibitReset := FALSE, bInternalReset := FALSE, aAlarmsSettings := gMessage.aAlarmsSettings, nAlarmIndex := nAlarmIndex, sMsgInfo := gMessage.stAlarmTable.aMsgHMI[nAlarmIndex], stMsgAux := gMessage.stAlarmTable.aMsgAux[nAlarmIndex]);

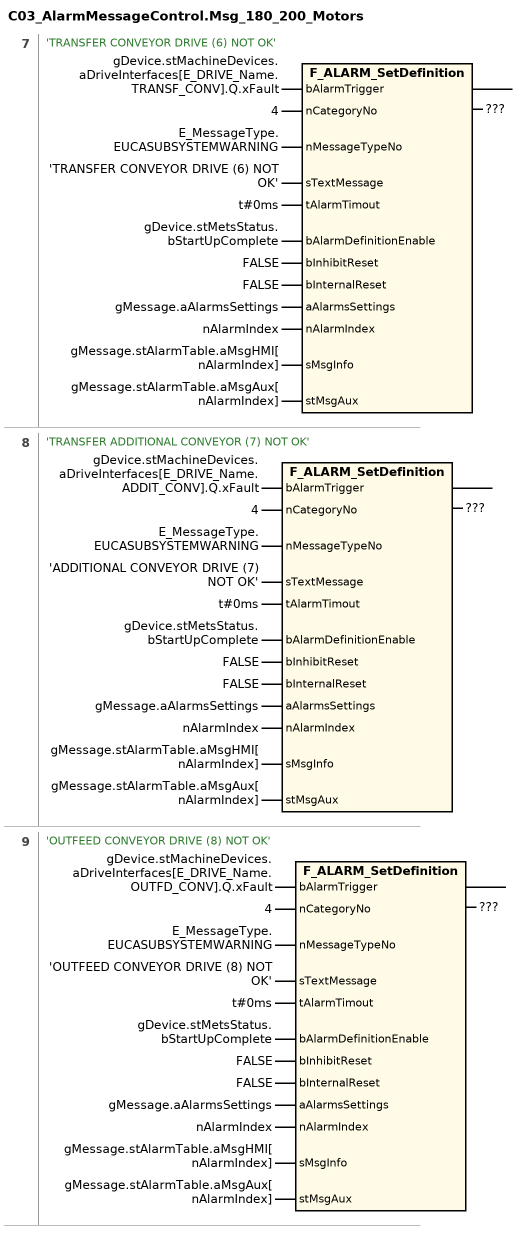
// NETWORK 7
// 'TRANSFER CONVEYOR DRIVE (6) NOT OK'
F_ALARM_SetDefinition(bAlarmTrigger := gDevice.stMachineDevices.aDriveInterfaces[E_DRIVE_Name.TRANSF_CONV].Q.xFault, nCategoryNo := 4, nMessageTypeNo := E_MessageType.EUCASUBSYSTEMWARNING, sTextMessage := 'TRANSFER CONVEYOR DRIVE (6) NOT OK', tAlarmTimout := t#0ms, bAlarmDefinitionEnable := gDevice.stMetsStatus.bStartUpComplete, bInhibitReset := FALSE, bInternalReset := FALSE, aAlarmsSettings := gMessage.aAlarmsSettings, nAlarmIndex := nAlarmIndex, sMsgInfo := gMessage.stAlarmTable.aMsgHMI[nAlarmIndex], stMsgAux := gMessage.stAlarmTable.aMsgAux[nAlarmIndex]);

// NETWORK 8
// 'TRANSFER ADDITIONAL CONVEYOR (7) NOT OK'
F_ALARM_SetDefinition(bAlarmTrigger := gDevice.stMachineDevices.aDriveInterfaces[E_DRIVE_Name.ADDIT_CONV].Q.xFault, nCategoryNo := 4, nMessageTypeNo := E_MessageType.EUCASUBSYSTEMWARNING, sTextMessage := 'ADDITIONAL CONVEYOR DRIVE (7) NOT OK', tAlarmTimout := t#0ms, bAlarmDefinitionEnable := gDevice.stMetsStatus.bStartUpComplete, bInhibitReset := FALSE, bInternalReset := FALSE, aAlarmsSettings := gMessage.aAlarmsSettings, nAlarmIndex := nAlarmIndex, sMsgInfo := gMessage.stAlarmTable.aMsgHMI[nAlarmIndex], stMsgAux := gMessage.stAlarmTable.aMsgAux[nAlarmIndex]);

// NETWORK 9
// 'OUTFEED CONVEYOR DRIVE (8) NOT OK'
F_ALARM_SetDefinition(bAlarmTrigger := gDevice.stMachineDevices.aDriveInterfaces[E_DRIVE_Name.OUTFD_CONV].Q.xFault, nCategoryNo := 4, nMessageTypeNo := E_MessageType.EUCASUBSYSTEMWARNING, sTextMessage := 'OUTFEED CONVEYOR DRIVE (8) NOT OK', tAlarmTimout := t#0ms, bAlarmDefinitionEnable := gDevice.stMetsStatus.bStartUpComplete, bInhibitReset := FALSE, bInternalReset := FALSE, aAlarmsSettings := gMessage.aAlarmsSettings, nAlarmIndex := nAlarmIndex, sMsgInfo := gMessage.stAlarmTable.aMsgHMI[nAlarmIndex], stMsgAux := gMessage.stAlarmTable.aMsgAux[nAlarmIndex]);

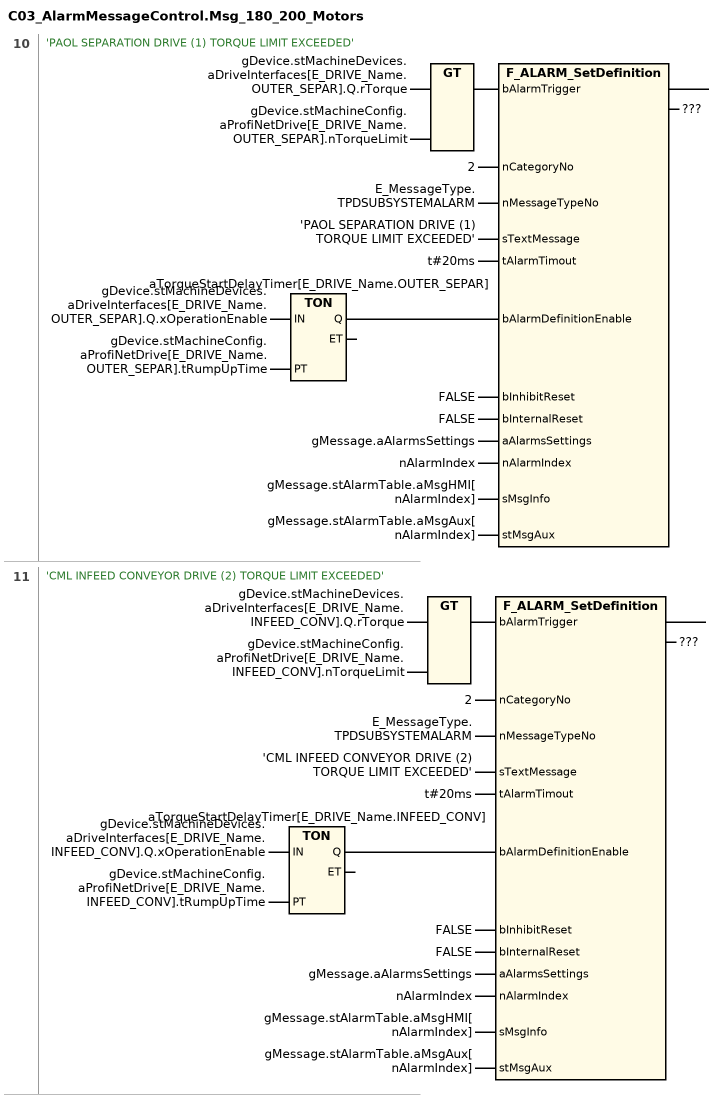
// NETWORK 10
// 'PAOL SEPARATION DRIVE (1) TORQUE LIMIT EXCEEDED'
aTorqueStartDelayTimer[E_DRIVE_Name.OUTER_SEPAR](IN := gDevice.stMachineDevices.aDriveInterfaces[E_DRIVE_Name.OUTER_SEPAR].Q.xOperationEnable, PT := gDevice.stMachineConfig.aProfiNetDrive[E_DRIVE_Name.OUTER_SEPAR].tRumpUpTime); // TON
F_ALARM_SetDefinition(bAlarmTrigger := gDevice.stMachineDevices.aDriveInterfaces[E_DRIVE_Name.OUTER_SEPAR].Q.rTorque > gDevice.stMachineConfig.aProfiNetDrive[E_DRIVE_Name.OUTER_SEPAR].nTorqueLimit, nCategoryNo := 2, nMessageTypeNo := E_MessageType.TPDSUBSYSTEMALARM, sTextMessage := 'PAOL SEPARATION DRIVE (1) TORQUE LIMIT EXCEEDED', tAlarmTimout := t#20ms, bAlarmDefinitionEnable := aTorqueStartDelayTimer[E_DRIVE_Name.OUTER_SEPAR].Q, bInhibitReset := FALSE, bInternalReset := FALSE, aAlarmsSettings := gMessage.aAlarmsSettings, nAlarmIndex := nAlarmIndex, sMsgInfo := gMessage.stAlarmTable.aMsgHMI[nAlarmIndex], stMsgAux := gMessage.stAlarmTable.aMsgAux[nAlarmIndex]);

// NETWORK 11
// 'CML INFEED CONVEYOR DRIVE (2) TORQUE LIMIT EXCEEDED'
aTorqueStartDelayTimer[E_DRIVE_Name.INFEED_CONV](IN := gDevice.stMachineDevices.aDriveInterfaces[E_DRIVE_Name.INFEED_CONV].Q.xOperationEnable, PT := gDevice.stMachineConfig.aProfiNetDrive[E_DRIVE_Name.INFEED_CONV].tRumpUpTime); // TON
F_ALARM_SetDefinition(bAlarmTrigger := gDevice.stMachineDevices.aDriveInterfaces[E_DRIVE_Name.INFEED_CONV].Q.rTorque > gDevice.stMachineConfig.aProfiNetDrive[E_DRIVE_Name.INFEED_CONV].nTorqueLimit, nCategoryNo := 2, nMessageTypeNo := E_MessageType.TPDSUBSYSTEMALARM, sTextMessage := 'CML INFEED CONVEYOR DRIVE (2) TORQUE LIMIT EXCEEDED', tAlarmTimout := t#20ms, bAlarmDefinitionEnable := aTorqueStartDelayTimer[E_DRIVE_Name.INFEED_CONV].Q, bInhibitReset := FALSE, bInternalReset := FALSE, aAlarmsSettings := gMessage.aAlarmsSettings, nAlarmIndex := nAlarmIndex, sMsgInfo := gMessage.stAlarmTable.aMsgHMI[nAlarmIndex], stMsgAux := gMessage.stAlarmTable.aMsgAux[nAlarmIndex]);

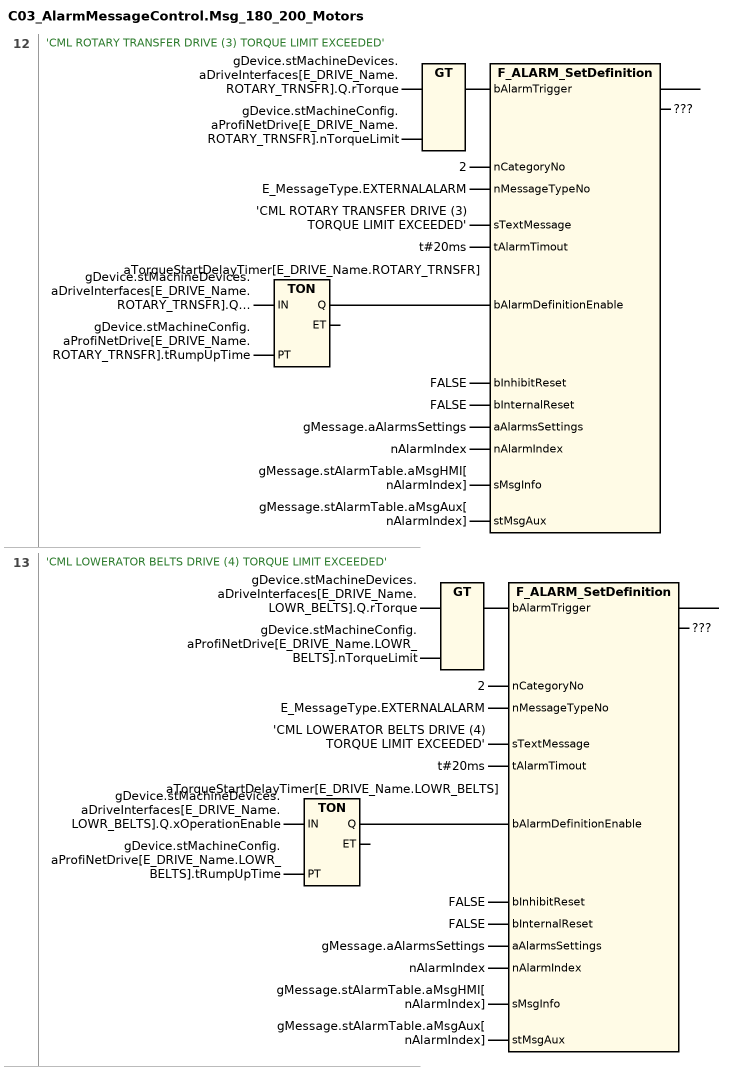
// NETWORK 12
// 'CML ROTARY TRANSFER DRIVE (3) TORQUE LIMIT EXCEEDED'
aTorqueStartDelayTimer[E_DRIVE_Name.ROTARY_TRNSFR](IN := gDevice.stMachineDevices.aDriveInterfaces[E_DRIVE_Name.ROTARY_TRNSFR].Q.xOperationEnable, PT := gDevice.stMachineConfig.aProfiNetDrive[E_DRIVE_Name.ROTARY_TRNSFR].tRumpUpTime); // TON
F_ALARM_SetDefinition(bAlarmTrigger := gDevice.stMachineDevices.aDriveInterfaces[E_DRIVE_Name.ROTARY_TRNSFR].Q.rTorque > gDevice.stMachineConfig.aProfiNetDrive[E_DRIVE_Name.ROTARY_TRNSFR].nTorqueLimit, nCategoryNo := 2, nMessageTypeNo := E_MessageType.EXTERNALALARM, sTextMessage := 'CML ROTARY TRANSFER DRIVE (3) TORQUE LIMIT EXCEEDED', tAlarmTimout := t#20ms, bAlarmDefinitionEnable := aTorqueStartDelayTimer[E_DRIVE_Name.ROTARY_TRNSFR].Q, bInhibitReset := FALSE, bInternalReset := FALSE, aAlarmsSettings := gMessage.aAlarmsSettings, nAlarmIndex := nAlarmIndex, sMsgInfo := gMessage.stAlarmTable.aMsgHMI[nAlarmIndex], stMsgAux := gMessage.stAlarmTable.aMsgAux[nAlarmIndex]);

// NETWORK 13
// 'CML LOWERATOR BELTS DRIVE (4) TORQUE LIMIT EXCEEDED'
aTorqueStartDelayTimer[E_DRIVE_Name.LOWR_BELTS](IN := gDevice.stMachineDevices.aDriveInterfaces[E_DRIVE_Name.LOWR_BELTS].Q.xOperationEnable, PT := gDevice.stMachineConfig.aProfiNetDrive[E_DRIVE_Name.LOWR_BELTS].tRumpUpTime); // TON
F_ALARM_SetDefinition(bAlarmTrigger := gDevice.stMachineDevices.aDriveInterfaces[E_DRIVE_Name.LOWR_BELTS].Q.rTorque > gDevice.stMachineConfig.aProfiNetDrive[E_DRIVE_Name.LOWR_BELTS].nTorqueLimit, nCategoryNo := 2, nMessageTypeNo := E_MessageType.EXTERNALALARM, sTextMessage := 'CML LOWERATOR BELTS DRIVE (4) TORQUE LIMIT EXCEEDED', tAlarmTimout := t#20ms, bAlarmDefinitionEnable := aTorqueStartDelayTimer[E_DRIVE_Name.LOWR_BELTS].Q, bInhibitReset := FALSE, bInternalReset := FALSE, aAlarmsSettings := gMessage.aAlarmsSettings, nAlarmIndex := nAlarmIndex, sMsgInfo := gMessage.stAlarmTable.aMsgHMI[nAlarmIndex], stMsgAux := gMessage.stAlarmTable.aMsgAux[nAlarmIndex]);

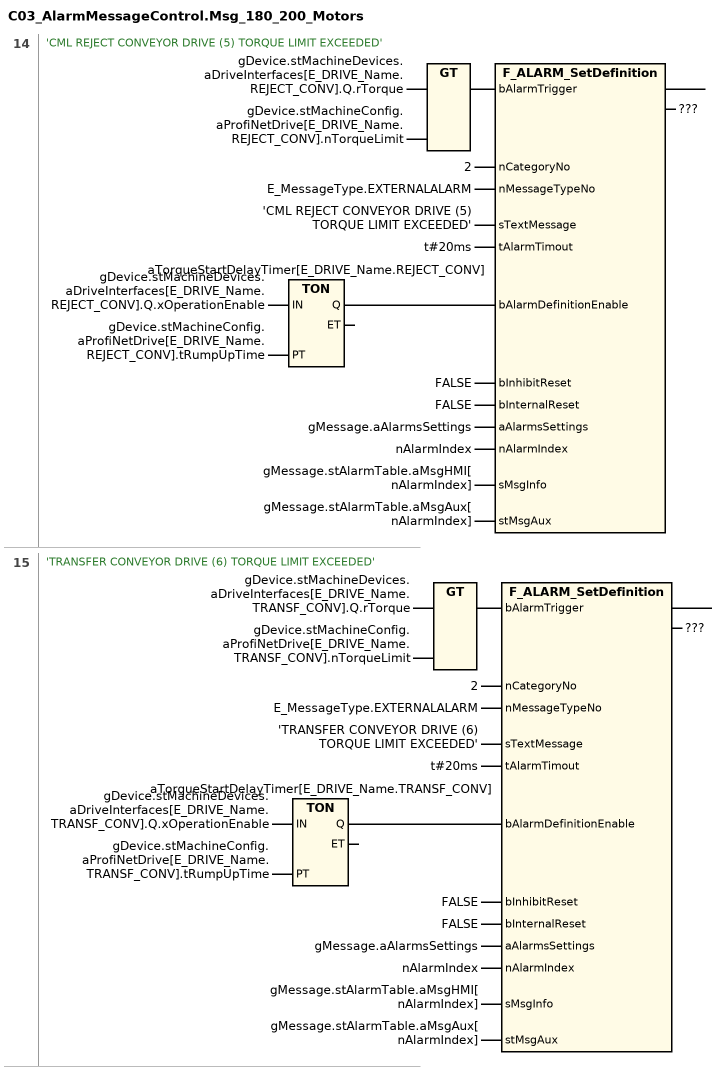
// NETWORK 14
// 'CML REJECT CONVEYOR DRIVE (5) TORQUE LIMIT EXCEEDED'
aTorqueStartDelayTimer[E_DRIVE_Name.REJECT_CONV](IN := gDevice.stMachineDevices.aDriveInterfaces[E_DRIVE_Name.REJECT_CONV].Q.xOperationEnable, PT := gDevice.stMachineConfig.aProfiNetDrive[E_DRIVE_Name.REJECT_CONV].tRumpUpTime); // TON
F_ALARM_SetDefinition(bAlarmTrigger := gDevice.stMachineDevices.aDriveInterfaces[E_DRIVE_Name.REJECT_CONV].Q.rTorque > gDevice.stMachineConfig.aProfiNetDrive[E_DRIVE_Name.REJECT_CONV].nTorqueLimit, nCategoryNo := 2, nMessageTypeNo := E_MessageType.EXTERNALALARM, sTextMessage := 'CML REJECT CONVEYOR DRIVE (5) TORQUE LIMIT EXCEEDED', tAlarmTimout := t#20ms, bAlarmDefinitionEnable := aTorqueStartDelayTimer[E_DRIVE_Name.REJECT_CONV].Q, bInhibitReset := FALSE, bInternalReset := FALSE, aAlarmsSettings := gMessage.aAlarmsSettings, nAlarmIndex := nAlarmIndex, sMsgInfo := gMessage.stAlarmTable.aMsgHMI[nAlarmIndex], stMsgAux := gMessage.stAlarmTable.aMsgAux[nAlarmIndex]);

// NETWORK 15
// 'TRANSFER CONVEYOR DRIVE (6) TORQUE LIMIT EXCEEDED'
aTorqueStartDelayTimer[E_DRIVE_Name.TRANSF_CONV](IN := gDevice.stMachineDevices.aDriveInterfaces[E_DRIVE_Name.TRANSF_CONV].Q.xOperationEnable, PT := gDevice.stMachineConfig.aProfiNetDrive[E_DRIVE_Name.TRANSF_CONV].tRumpUpTime); // TON
F_ALARM_SetDefinition(bAlarmTrigger := gDevice.stMachineDevices.aDriveInterfaces[E_DRIVE_Name.TRANSF_CONV].Q.rTorque > gDevice.stMachineConfig.aProfiNetDrive[E_DRIVE_Name.TRANSF_CONV].nTorqueLimit, nCategoryNo := 2, nMessageTypeNo := E_MessageType.EXTERNALALARM, sTextMessage := 'TRANSFER CONVEYOR DRIVE (6) TORQUE LIMIT EXCEEDED', tAlarmTimout := t#20ms, bAlarmDefinitionEnable := aTorqueStartDelayTimer[E_DRIVE_Name.TRANSF_CONV].Q, bInhibitReset := FALSE, bInternalReset := FALSE, aAlarmsSettings := gMessage.aAlarmsSettings, nAlarmIndex := nAlarmIndex, sMsgInfo := gMessage.stAlarmTable.aMsgHMI[nAlarmIndex], stMsgAux := gMessage.stAlarmTable.aMsgAux[nAlarmIndex]);

